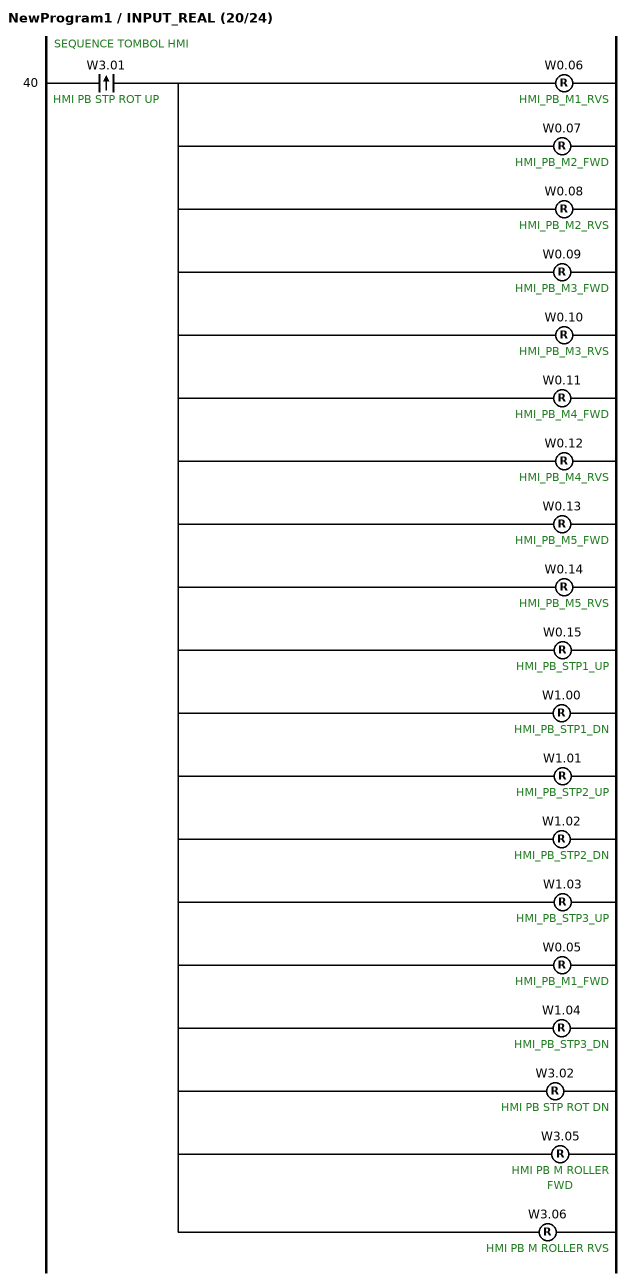
; [picture p48: NewProgram1 / INPUT_REAL, rungs 40-40]
; rung 40: SEQUENCE TOMBOL HMI
@LD W3.01  ; HMI PB STP ROT UP
RSET W0.06  ; HMI_PB_M1_RVS
RSET W0.07  ; HMI_PB_M2_FWD
RSET W0.08  ; HMI_PB_M2_RVS
RSET W0.09  ; HMI_PB_M3_FWD
RSET W0.10  ; HMI_PB_M3_RVS
RSET W0.11  ; HMI_PB_M4_FWD
RSET W0.12  ; HMI_PB_M4_RVS
RSET W0.13  ; HMI_PB_M5_FWD
RSET W0.14  ; HMI_PB_M5_RVS
RSET W0.15  ; HMI_PB_STP1_UP
RSET W1.00  ; HMI_PB_STP1_DN
RSET W1.01  ; HMI_PB_STP2_UP
RSET W1.02  ; HMI_PB_STP2_DN
RSET W1.03  ; HMI_PB_STP3_UP
RSET W0.05  ; HMI_PB_M1_FWD
RSET W1.04  ; HMI_PB_STP3_DN
RSET W3.02  ; HMI PB STP ROT DN
RSET W3.05  ; HMI PB M ROLLER FWD
RSET W3.06  ; HMI PB M ROLLER RVS

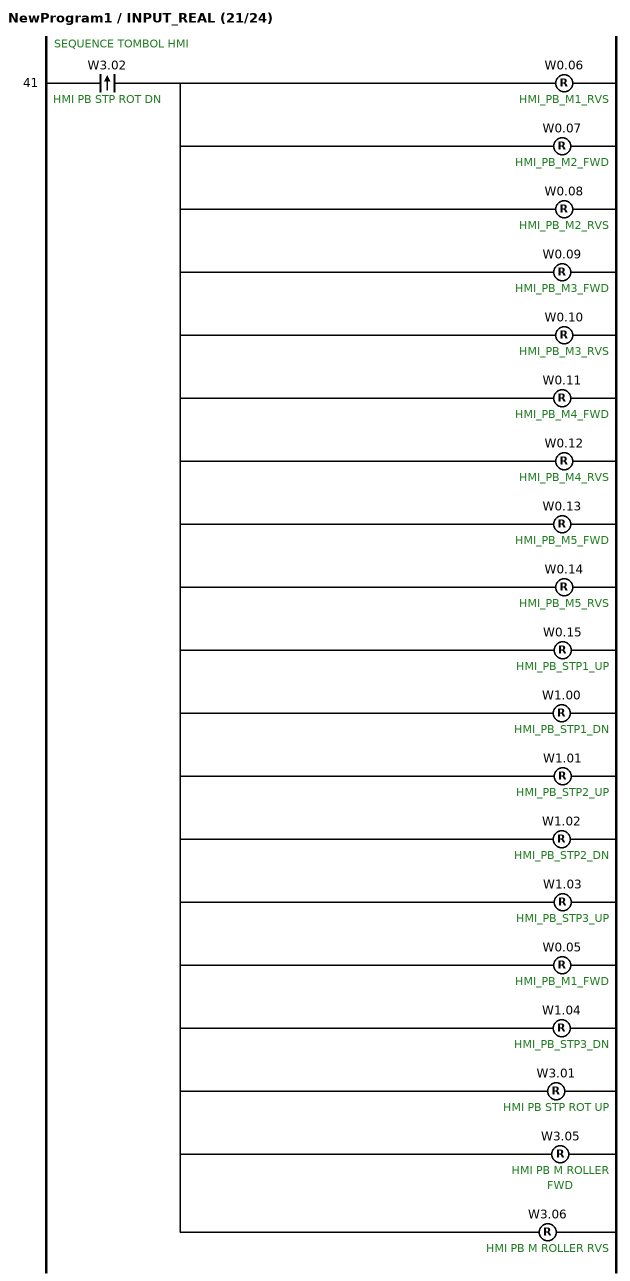
; rung 41: SEQUENCE TOMBOL HMI
@LD W3.02  ; HMI PB STP ROT DN
RSET W0.06  ; HMI_PB_M1_RVS
RSET W0.07  ; HMI_PB_M2_FWD
RSET W0.08  ; HMI_PB_M2_RVS
RSET W0.09  ; HMI_PB_M3_FWD
RSET W0.10  ; HMI_PB_M3_RVS
RSET W0.11  ; HMI_PB_M4_FWD
RSET W0.12  ; HMI_PB_M4_RVS
RSET W0.13  ; HMI_PB_M5_FWD
RSET W0.14  ; HMI_PB_M5_RVS
RSET W0.15  ; HMI_PB_STP1_UP
RSET W1.00  ; HMI_PB_STP1_DN
RSET W1.01  ; HMI_PB_STP2_UP
RSET W1.02  ; HMI_PB_STP2_DN
RSET W1.03  ; HMI_PB_STP3_UP
RSET W0.05  ; HMI_PB_M1_FWD
RSET W1.04  ; HMI_PB_STP3_DN
RSET W3.01  ; HMI PB STP ROT UP
RSET W3.05  ; HMI PB M ROLLER FWD
RSET W3.06  ; HMI PB M ROLLER RVS

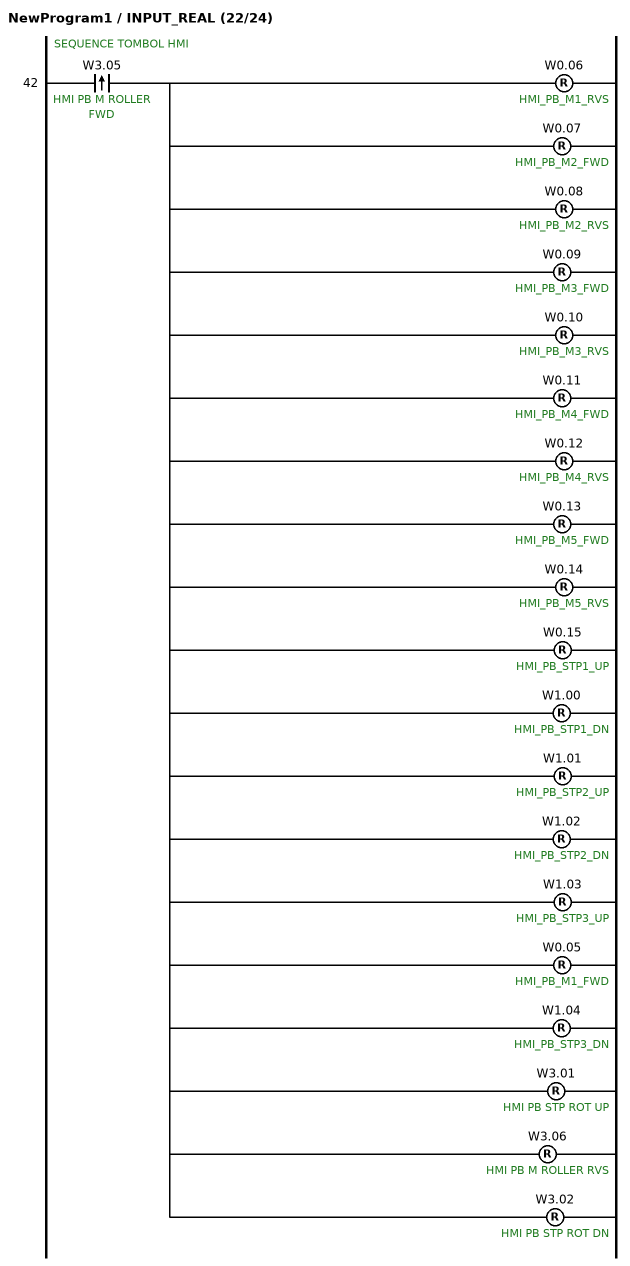
; rung 42: SEQUENCE TOMBOL HMI
@LD W3.05  ; HMI PB M ROLLER FWD
RSET W0.06  ; HMI_PB_M1_RVS
RSET W0.07  ; HMI_PB_M2_FWD
RSET W0.08  ; HMI_PB_M2_RVS
RSET W0.09  ; HMI_PB_M3_FWD
RSET W0.10  ; HMI_PB_M3_RVS
RSET W0.11  ; HMI_PB_M4_FWD
RSET W0.12  ; HMI_PB_M4_RVS
RSET W0.13  ; HMI_PB_M5_FWD
RSET W0.14  ; HMI_PB_M5_RVS
RSET W0.15  ; HMI_PB_STP1_UP
RSET W1.00  ; HMI_PB_STP1_DN
RSET W1.01  ; HMI_PB_STP2_UP
RSET W1.02  ; HMI_PB_STP2_DN
RSET W1.03  ; HMI_PB_STP3_UP
RSET W0.05  ; HMI_PB_M1_FWD
RSET W1.04  ; HMI_PB_STP3_DN
RSET W3.01  ; HMI PB STP ROT UP
RSET W3.06  ; HMI PB M ROLLER RVS
RSET W3.02  ; HMI PB STP ROT DN

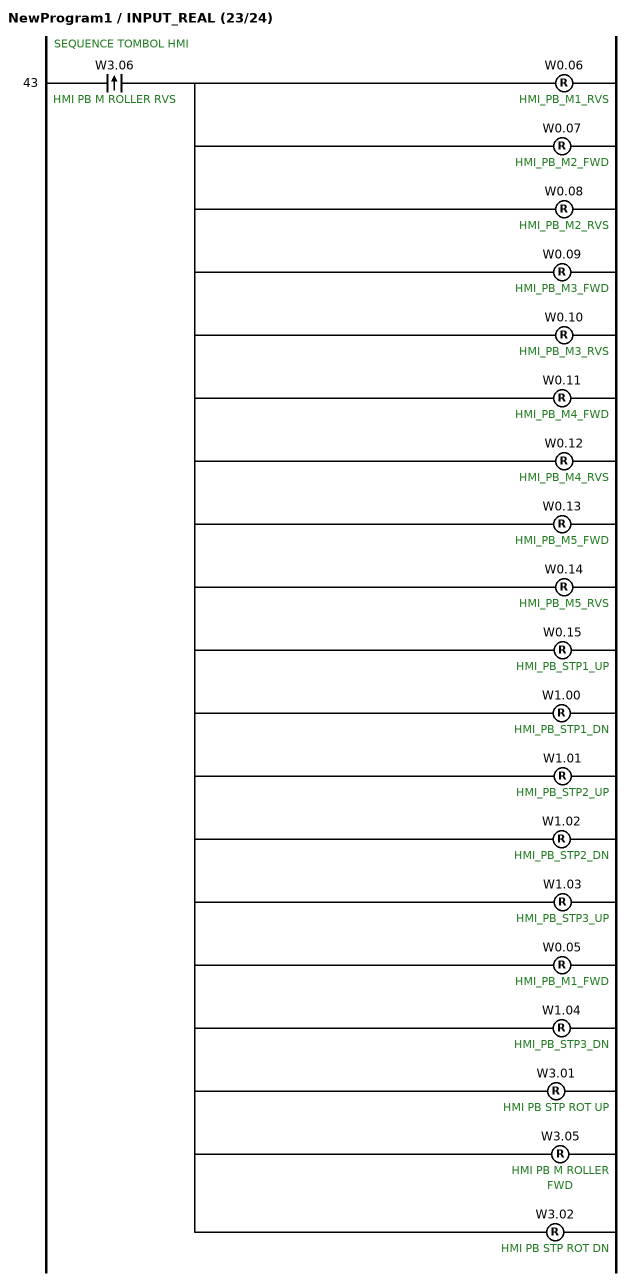
; rung 43: SEQUENCE TOMBOL HMI
@LD W3.06  ; HMI PB M ROLLER RVS
RSET W0.06  ; HMI_PB_M1_RVS
RSET W0.07  ; HMI_PB_M2_FWD
RSET W0.08  ; HMI_PB_M2_RVS
RSET W0.09  ; HMI_PB_M3_FWD
RSET W0.10  ; HMI_PB_M3_RVS
RSET W0.11  ; HMI_PB_M4_FWD
RSET W0.12  ; HMI_PB_M4_RVS
RSET W0.13  ; HMI_PB_M5_FWD
RSET W0.14  ; HMI_PB_M5_RVS
RSET W0.15  ; HMI_PB_STP1_UP
RSET W1.00  ; HMI_PB_STP1_DN
RSET W1.01  ; HMI_PB_STP2_UP
RSET W1.02  ; HMI_PB_STP2_DN
RSET W1.03  ; HMI_PB_STP3_UP
RSET W0.05  ; HMI_PB_M1_FWD
RSET W1.04  ; HMI_PB_STP3_DN
RSET W3.01  ; HMI PB STP ROT UP
RSET W3.05  ; HMI PB M ROLLER FWD
RSET W3.02  ; HMI PB STP ROT DN

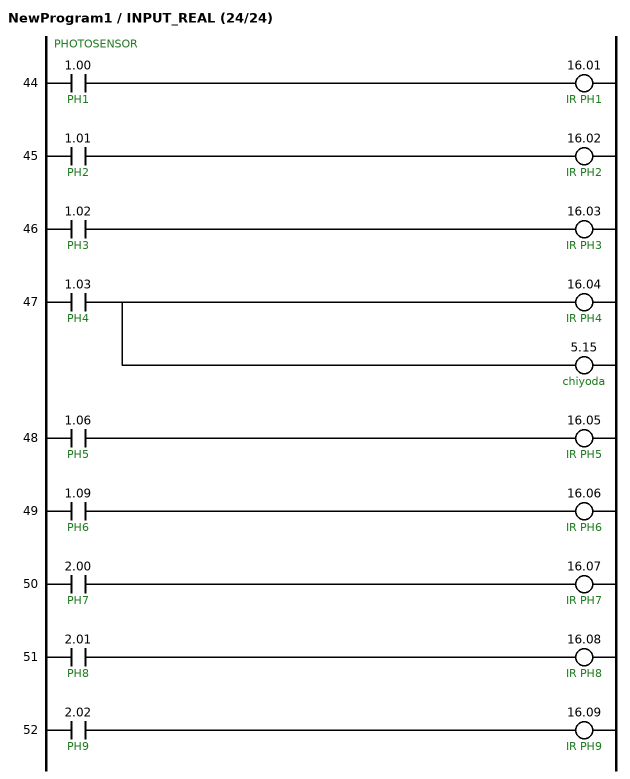
; rung 44: PHOTOSENSOR
LD 1.00  ; PH1
OUT 16.01  ; IR PH1
; rung 45
LD 1.01  ; PH2
OUT 16.02  ; IR PH2
; rung 46
LD 1.02  ; PH3
OUT 16.03  ; IR PH3
; rung 47
LD 1.03  ; PH4
OUT 16.04  ; IR PH4
OUT 5.15  ; chiyoda
; rung 48
LD 1.06  ; PH5
OUT 16.05  ; IR PH5
; rung 49
LD 1.09  ; PH6
OUT 16.06  ; IR PH6
; rung 50
LD 2.00  ; PH7
OUT 16.07  ; IR PH7
; rung 51
LD 2.01  ; PH8
OUT 16.08  ; IR PH8
; rung 52
LD 2.02  ; PH9
OUT 16.09  ; IR PH9

### Section END
; rung 0
END(001)

## Function block DATAMOVEMENT
VAR_INPUT
  DataIn1 : WORD;
  DataIn2 : WORD;
  DataIn3 : WORD;
  DataIn4 : WORD;
  DataIn5 : WORD;
  ENABLING : BOOL;
END_VAR
VAR_OUTPUT
  DataOut1 : WORD;
  DataOut2 : WORD;
END_VAR
IF EN THEN
	
IF ENABLING = TRUE AND  DataIn1 = 16#0266 AND DataIn2 = 16#6630 AND DataIn5 = 16#3030 THEN
	DataOut1 := DataIn4;
	DataOut2 :=  DataIn3;
	END_IF;
END_IF;

## Function block FOR
VAR_INPUT
  DATA_INPUT : DWORD;
  DATA_INDIRECT : INT;
  INCOMING_DATA_RFID : DWORD;
  CAN_COMFIRMED : BOOL;
END_VAR
VAR_OUTPUT
  CONFIRM : BOOL;
END_VAR
VAR
  d : INT;
  Array_boy : ARRAY[0..186] OF DWORD;
END_VAR
IF EN THEN 
	(* INITIALIATION*)
Array_boy [DATA_INDIRECT] := DATA_INPUT;

FOR d := 0 TO 187 DO
	IF Array_boy [DATA_INDIRECT] = INCOMING_DATA_RFID AND CAN_COMFIRMED = FALSE
		THEN
		CONFIRM := TRUE ;
	ELSE 
		CONFIRM := FALSE ;
	END_IF;
END_FOR;
END_IF;

## Function block NO_BLOWING
VAR_INPUT
  RETAIN MEMORY_1 : DWORD;
  RETAIN MEMORY_2 : DWORD;
  RETAIN MEMORY_3 : DWORD;
  RETAIN MEMORY_4 : DWORD;
  RETAIN MEMORY_5 : DWORD;
  RETAIN MEMORY_6 : DWORD;
  RETAIN MEMORY_7 : DWORD;
  RETAIN MEMORY_8 : DWORD;
  RETAIN MEMORY_9 : DWORD;
  RETAIN MEMORY_10 : DWORD;
  DATA_INCOMING : DWORD;
END_VAR
VAR_OUTPUT
  NO_BLOWING_CONFIRM : BOOL;
END_VAR

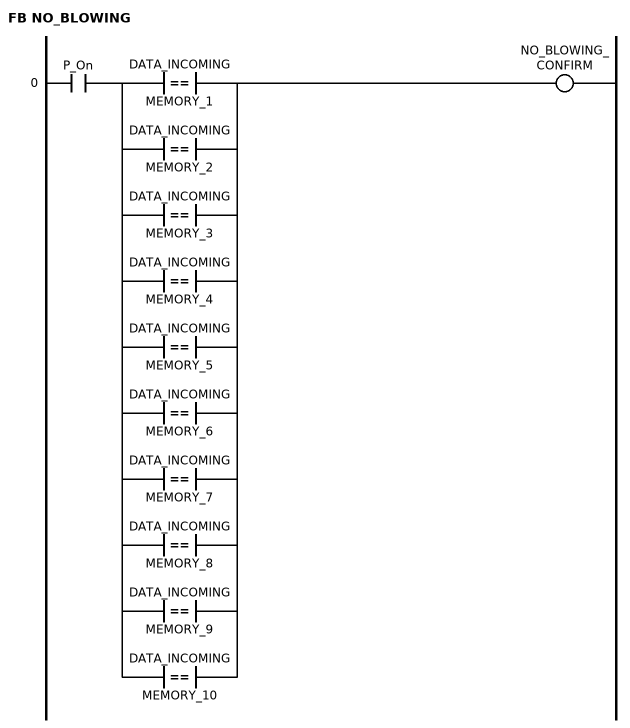
; rung 0
LD P_On
LD=(300) DATA_INCOMING MEMORY_1
OR=(300) DATA_INCOMING MEMORY_2
OR=(300) DATA_INCOMING MEMORY_3
OR=(300) DATA_INCOMING MEMORY_4
OR=(300) DATA_INCOMING MEMORY_5
OR=(300) DATA_INCOMING MEMORY_6
OR=(300) DATA_INCOMING MEMORY_7
OR=(300) DATA_INCOMING MEMORY_8
OR=(300) DATA_INCOMING MEMORY_9
OR=(300) DATA_INCOMING MEMORY_10
ANDLD
OUT NO_BLOWING_CONFIRM